// Mitsubishi GX Works2 project: Test   PLC: Q00J

PROGRAM MAIN
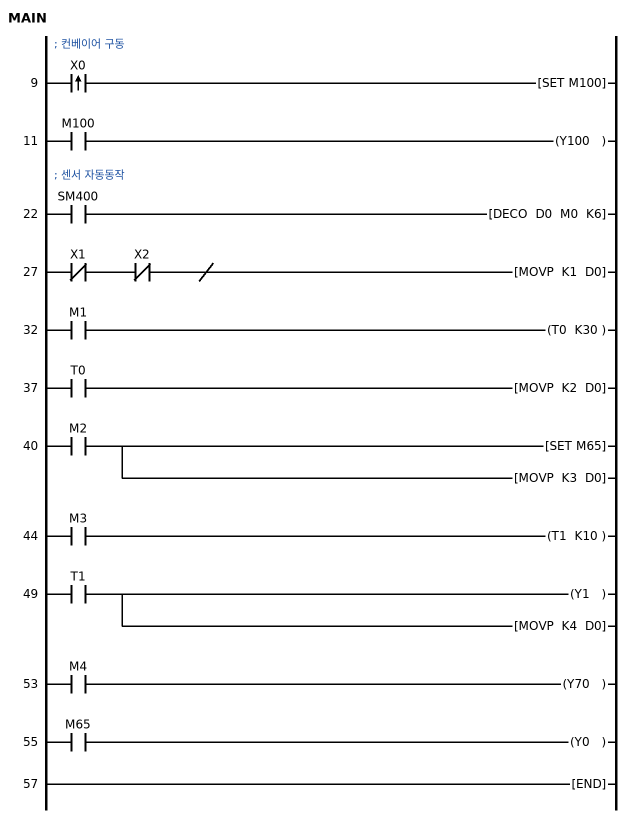
; 컨베이어 구동
9     LDP     X0
      SET     M100
11    LD      M100
      OUT     Y100
; 센서 자동동작
22    LD      SM400
      DECO    D0 M0 K6
27    LDI     X1
      ANI     X2
      INV
      MOVP    K1 D0
32    LD      M1
      OUT     T0 K30
37    LD      T0
      MOVP    K2 D0
40    LD      M2
      SET     M65
      MOVP    K3 D0
44    LD      M3
      OUT     T1 K10
49    LD      T1
      OUT     Y1
      MOVP    K4 D0
53    LD      M4
      OUT     Y70
55    LD      M65
      OUT     Y0
57    END
END_PROGRAM
